TYPE ST_GantryProdPar_Org :
STRUCT
	PositionHorizontalPickup			: LREAL;
	PositionHorizontalDropOff			: LREAL;
	PositionVerticalPickup				: LREAL;
	PositionVerticalDropOff				: LREAL;
	
	BlowOffTime							: TIME;
	
END_STRUCT
END_TYPE

(* stored: Version 1.1.0.1, ProductVersion 3.1.4020.12
   DUT ST_GantryProdPar_Org: Id {9a55c172-9271-49e2-aede-afa42768ef23} *)
